{attribute 'GeneratedUsingTerminal: EK1100-0000-0018'}
{attribute addProperty BoxType "EK1100-0000-0018"}
{attribute addProperty Id "Beckhoff_EP1xxxEK1122Beckhoff_EP1xxxEK1122_F9185EC31740"}
{attribute addProperty CRC "1828796328"}
{attribute addProperty Size "1740"}
TYPE Beckhoff_EP1xxx_6D0137A8 EXTENDS EK1100_AB5A9467 :
STRUCT
	{attribute addProperty Name "Beckhoff_EP1xxxEK1122"}
	Beckhoff_EP1xxxEK1122 : Beckhoff_EP1xxxEK1122_F9185EC3;
END_STRUCT
END_TYPE

(* stored: Version 1.2.0.0, ProductVersion 3.1.4024.9
   DUT Beckhoff_EP1xxx_6D0137A8: Id {95393976-16cb-49ca-8e6f-b5d8106fe2aa} *)
